Staubli VAL3: decodeShareReal.pgx

public program decodeShareReal(num& x_nStatus (dimensions=1), num& x_nValue (dimensions=1), num& x_nDWordBody[] (dimensions=2), num x_nRowIndex (dimensions=1))
  local num l_nDWordBytes[4]
begin
  if x_nStatus<0
    return
  endIf
  x_nStatus=-1
  call getRow(l_nDWordBytes,x_nDWordBody,x_nRowIndex)
  x_nStatus=fromBinary(l_nDWordBytes,4,"4.0l",x_nValue)
  if x_nStatus<0
    putln("Failed to decode shared float at index "+toString("",x_nRowIndex)+" with status "+toString("",x_nStatus))
  endIf
end
